LIN {X 0,Y 62.23,Z 1055.519,A -85,B 0,C 180,E1 2367.907,E2 2367.907} C_VEL
LIN {X 0,Y 81.235,Z 1051.075,A -85,B 0,C 180,E1 2356.249,E2 2356.249} C_VEL
LIN {X 0,Y 105.062,Z 1044.254,A -85,B 0,C 180,E1 2348.201,E2 2348.201} C_VEL
LIN {X 0,Y 125.272,Z 1037.346,A -85,B 0,C 180,E1 2343.877,E2 2343.877} C_VEL
LIN {X 0,Y 146.99,Z 1028.752,A -85,B 0,C 180,E1 2340.583,E2 2340.583} C_VEL
LIN {X 0,Y 167.827,Z 1019.239,A -85,B 0,C 180,E1 2338.199,E2 2338.199} C_VEL
LIN {X 0,Y 144.434,Z 1029.702,A -85,B 0,C 180,E1 2335.468,E2 2335.468} C_VEL
LIN {X 0,Y 124.116,Z 1037.572,A -85,B 0,C 180,E1 2332.261,E2 2332.261} C_VEL
LIN {X 0,Y 100.607,Z 1045.395,A -85,B 0,C 180,E1 2326.899,E2 2326.899} C_VEL
LIN {X 0,Y 78.368,Z 1051.328,A -85,B 0,C 180,E1 2318.652,E2 2318.652} C_VEL
LIN {X 0,Y 61.249,Z 1055.193,A -85,B 0,C 180,E1 2307.403,E2 2307.403} C_VEL
LIN {X 0,Y 47.043,Z 1058.07,A -85,B 0,C 180,E1 2288.052,E2 2288.052} C_VEL
LIN {X 0,Y 40.29,Z 1059.695,A -85,B 0,C 180,E1 2260.004,E2 2260.004} C_VEL
LIN {X 0,Y 39.914,Z 1059.95,A -85,B 0,C 180,E1 2244.249,E2 2244.249} C_VEL
LIN {X 0,Y 41.264,Z 1060.011,A -85,B 0,C 180,E1 2225.673,E2 2225.673} C_VEL
LIN {X 0,Y 49.39,Z 1059.265,A -85,B 0,C 180,E1 2201.491,E2 2201.491} C_VEL
LIN {X 0,Y 63.805,Z 1057.416,A -85,B 0,C 180,E1 2184.643,E2 2184.643} C_VEL
LIN {X 0,Y 84.152,Z 1053.993,A -85,B 0,C 180,E1 2173.014,E2 2173.014} C_VEL
LIN {X 0,Y 108.886,Z 1048.344,A -85,B 0,C 180,E1 2165.269,E2 2165.269} C_VEL
LIN {X 0,Y 130.008,Z 1042.364,A -85,B 0,C 180,E1 2161.081,E2 2161.081} C_VEL
LIN {X 0,Y 145.554,Z 1037.228,A -85,B 0,C 180,E1 2158.77,E2 2158.77} C_VEL
LIN {X 0,Y 123.274,Z 1044.544,A -85,B 0,C 180,E1 2155.348,E2 2155.348} C_VEL
LIN {X 0,Y 99.855,Z 1050.86,A -85,B 0,C 180,E1 2150.04,E2 2150.04} C_VEL
LIN {X 0,Y 92.672,Z 1052.424,A -85,B 0,C 180,E1 2148.54,E2 2148.54} C_VEL
LIN {X 0,Y 72.154,Z 1056.236,A -85,B 0,C 180,E1 2145.682,E2 2145.682} C_VEL
LIN {X 0,Y 66.123,Z 1057.108,A -85,B 0,C 180,E1 2143.439,E2 2143.439} C_VEL
LIN {X 0,Y 46.36,Z 1059.586,A -85,B 0,C 180,E1 2127.261,E2 2127.261} C_VEL
LIN {X 0,Y 35.013,Z 1060.577,A -85,B 0,C 180,E1 2102.861,E2 2102.861} C_VEL
LIN {X 0,Y 31.935,Z 1060.688,A -85,B 0,C 180,E1 2077.195,E2 2077.195} C_VEL
LIN {X 0,Y 31.933,Z 1060.508,A -85,B 0,C 180,E1 2062.806,E2 2062.806} C_VEL
LIN {X 0,Y 35.788,Z 1059.542,A -85,B 0,C 180,E1 2034.076,E2 2034.076} C_VEL
LIN {X 0,Y 50.744,Z 1057.023,A -85,B 0,C 180,E1 2007.539,E2 2007.539} C_VEL
LIN {X 0,Y 71.957,Z 1052.634,A -85,B 0,C 180,E1 1993.424,E2 1993.424} C_VEL
LIN {X 0,Y 91.601,Z 1047.732,A -85,B 0,C 180,E1 1986.625,E2 1986.625} C_VEL
LIN {X 0,Y 116.023,Z 1040.405,A -85,B 0,C 180,E1 1981.451,E2 1981.451} C_VEL
LIN {X 0,Y 139.32,Z 1031.761,A -85,B 0,C 180,E1 1978.189,E2 1978.189} C_VEL
LIN {X 0,Y 114.491,Z 1040.77,A -85,B 0,C 180,E1 1974.617,E2 1974.617} C_VEL
LIN {X 0,Y 91.487,Z 1047.54,A -85,B 0,C 180,E1 1969.616,E2 1969.616} C_VEL
LIN {X 0,Y 71.294,Z 1052.467,A -85,B 0,C 180,E1 1962.493,E2 1962.493} C_VEL
LIN {X 0,Y 49.02,Z 1056.839,A -85,B 0,C 180,E1 1946.75,E2 1946.75} C_VEL
LIN {X 0,Y 35.858,Z 1058.993,A -85,B 0,C 180,E1 1921.992,E2 1921.992} C_VEL
LIN {X 0,Y 31.97,Z 1059.896,A -85,B 0,C 180,E1 1893.586,E2 1893.586} C_VEL
LIN {X 0,Y 32.157,Z 1060.129,A -85,B 0,C 180,E1 1875.596,E2 1875.596} C_VEL
LIN {X 0,Y 39.331,Z 1059.836,A -85,B 0,C 180,E1 1842.502,E2 1842.502} C_VEL
LIN {X 0,Y 57.397,Z 1057.92,A -85,B 0,C 180,E1 1819.827,E2 1819.827} C_VEL
LIN {X 0,Y 77.014,Z 1054.988,A -85,B 0,C 180,E1 1809.347,E2 1809.347} C_VEL
LIN {X 0,Y 101.426,Z 1050.147,A -85,B 0,C 180,E1 1802.26,E2 1802.26} C_VEL
LIN {X 0,Y 120.013,Z 1045.405,A -85,B 0,C 180,E1 1798.786,E2 1798.786} C_VEL
LIN {X 0,Y 94.543,Z 1051.731,A -85,B 0,C 180,E1 1793.795,E2 1793.795} C_VEL
LIN {X 0,Y 73.855,Z 1055.787,A -85,B 0,C 180,E1 1787.103,E2 1787.103} C_VEL
LIN {X 0,Y 66.123,Z 1057.108,A -85,B 0,C 180,E1 1783.439,E2 1783.439} C_VEL
LIN {X 0,Y 59.161,Z 1057.998,A -85,B 0,C 180,E1 1780.392,E2 1780.392} C_VEL
LIN {X 0,Y 38.812,Z 1060.018,A -85,B 0,C 180,E1 1771.206,E2 1771.206} C_VEL
LIN {X 0,Y 34.014,Z 1060.279,A -85,B 0,C 180,E1 1765.205,E2 1765.205} C_VEL
LIN {X 0,Y 24.195,Z 1060.648,A -85,B 0,C 180,E1 1724.358,E2 1724.358} C_VEL
LIN {X 0,Y 23.898,Z 1060.472,A -85,B 0,C 180,E1 1705.201,E2 1705.201} C_VEL
LIN {X 0,Y 27.039,Z 1059.798,A -85,B 0,C 180,E1 1673.725,E2 1673.725} C_VEL
LIN {X 0,Y 39.211,Z 1058.087,A -85,B 0,C 180,E1 1646.813,E2 1646.813} C_VEL
LIN {X 0,Y 57.327,Z 1055.125,A -85,B 0,C 180,E1 1632.383,E2 1632.383} C_VEL
LIN {X 0,Y 81.873,Z 1049.995,A -85,B 0,C 180,E1 1623.501,E2 1623.501} C_VEL
LIN {X 0,Y 106.013,Z 1043.342,A -85,B 0,C 180,E1 1618.741,E2 1618.741} C_VEL
LIN {X 0,Y 109.795,Z 1042.185,A -85,B 0,C 180,E1 1618.138,E2 1618.138} C_VEL
LIN {X 0,Y 88.425,Z 1048.176,A -85,B 0,C 180,E1 1614.313,E2 1614.313} C_VEL
LIN {X 0,Y 64.607,Z 1053.606,A -85,B 0,C 180,E1 1607.164,E2 1607.164} C_VEL
LIN {X 0,Y 41.807,Z 1057.387,A -85,B 0,C 180,E1 1592.24,E2 1592.24} C_VEL
LIN {X 0,Y 28.279,Z 1059.218,A -85,B 0,C 180,E1 1566.946,E2 1566.946} C_VEL
LIN {X 0,Y 23.986,Z 1059.979,A -85,B 0,C 180,E1 1534.781,E2 1534.781} C_VEL
LIN {X 0,Y 24.237,Z 1060.188,A -85,B 0,C 180,E1 1513.214,E2 1513.214} C_VEL
LIN {X 0,Y 32.914,Z 1059.953,A -85,B 0,C 180,E1 1474.891,E2 1474.891} C_VEL
LIN {X 0,Y 54.21,Z 1058.087,A -85,B 0,C 180,E1 1452.156,E2 1452.156} C_VEL
LIN {X 0,Y 75.123,Z 1055.192,A -85,B 0,C 180,E1 1443.382,E2 1443.382} C_VEL
LIN {X 0,Y 93.785,Z 1051.742,A -85,B 0,C 180,E1 1438.8,E2 1438.8} C_VEL
LIN {X 0,Y 72.457,Z 1055.741,A -85,B 0,C 180,E1 1433.509,E2 1433.509} C_VEL
LIN {X 0,Y 48.416,Z 1059.029,A -85,B 0,C 180,E1 1421.806,E2 1421.806} C_VEL
LIN {X 0,Y 34.014,Z 1060.279,A -85,B 0,C 180,E1 1405.205,E2 1405.205} C_VEL
LIN {X 0,Y 28.476,Z 1060.509,A -85,B 0,C 180,E1 1395.118,E2 1395.118} C_VEL
LIN {X 0,Y 21.095,Z 1060.68,A -85,B 0,C 180,E1 1377.104,E2 1377.104} C_VEL
LIN {X 0,Y 16.944,Z 1060.254,A -85,B 0,C 180,E1 1322.989,E2 1322.989} C_VEL
LIN {X 0,Y 31.831,Z 1058.564,A -85,B 0,C 180,E1 1279.547,E2 1279.547} C_VEL
LIN {X 0,Y 52.569,Z 1055.608,A -85,B 0,C 180,E1 1265.457,E2 1265.457} C_VEL
LIN {X 0,Y 73.999,Z 1051.54,A -85,B 0,C 180,E1 1259.166,E2 1259.166} C_VEL
LIN {X 0,Y 79.035,Z 1050.485,A -85,B 0,C 180,E1 1258.084,E2 1258.084} C_VEL
LIN {X 0,Y 55.552,Z 1055.004,A -85,B 0,C 180,E1 1251.869,E2 1251.869} C_VEL
LIN {X 0,Y 36.013,Z 1057.824,A -85,B 0,C 180,E1 1240.733,E2 1240.733} C_VEL
LIN {X 0,Y 20.45,Z 1059.511,A -85,B 0,C 180,E1 1213.196,E2 1213.196} C_VEL
LIN {X 0,Y 15.91,Z 1060.107,A -85,B 0,C 180,E1 1169.998,E2 1169.998} C_VEL
LIN {X 0,Y 18.067,Z 1060.358,A -85,B 0,C 180,E1 1132.498,E2 1132.498} C_VEL
LIN {X 0,Y 35.082,Z 1059.66,A -85,B 0,C 180,E1 1094.289,E2 1094.289} C_VEL
LIN {X 0,Y 56.034,Z 1057.808,A -85,B 0,C 180,E1 1082.17,E2 1082.17} C_VEL
LIN {X 0,Y 66.796,Z 1056.536,A -85,B 0,C 180,E1 1078.887,E2 1078.887} C_VEL
LIN {X 0,Y 41.792,Z 1059.315,A -85,B 0,C 180,E1 1068.795,E2 1068.795} C_VEL
LIN {X 0,Y 23.803,Z 1060.403,A -85,B 0,C 180,E1 1047.156,E2 1047.156} C_VEL
LIN {X 0,Y 16.114,Z 1060.522,A -85,B 0,C 180,E1 1004.372,E2 1004.372} C_VEL
LIN {X 0,Y 15.989,Z 1060.366,A -85,B 0,C 180,E1 979.189,E2 979.189} C_VEL
LIN {X 0,Y 16.944,Z 1060.254,A -85,B 0,C 180,E1 962.989,E2 962.989} C_VEL
LIN {X 0,Y 19.569,Z 1059.953,A -85,B 0,C 180,E1 941.806,E2 941.806} C_VEL
LIN {X 0,Y 26.288,Z 1059.023,A -85,B 0,C 180,E1 915.615,E2 915.615} C_VEL
LIN {X 0,Y 35.66,Z 1057.813,A -85,B 0,C 180,E1 902.3,E2 902.3} C_VEL
LIN {X 0,Y 39.85,Z 1057.312,A -85,B 0,C 180,E1 900.013,E2 900.013} C_VEL
LIN {X 0,Y 45.651,Z 1056.586,A -85,B 0,C 180,E1 898.004,E2 898.004} C_VEL
LIN {X 0,Y 21.184,Z 1059.185,A -85,B 0,C 180,E1 883.548,E2 883.548} C_VEL
LIN {X 0,Y 8.405,Z 1060.123,A -85,B 0,C 180,E1 830.907,E2 830.907} C_VEL
LIN {X 0,Y 8.481,Z 1060.284,A -85,B 0,C 180,E1 781.86,E2 781.86} C_VEL
LIN {X 0,Y 21.347,Z 1060.227,A -85,B 0,C 180,E1 730.374,E2 730.374} C_VEL
LIN {X 0,Y 37.624,Z 1059.486,A -85,B 0,C 180,E1 718.952,E2 718.952} C_VEL
LIN {X 0,Y 18.721,Z 1060.378,A -85,B 0,C 180,E1 704.025,E2 704.025} C_VEL
LIN {X 0,Y 8.236,Z 1060.418,A -85,B 0,C 180,E1 651.362,E2 651.362} C_VEL
LIN {X 0,Y 8.234,Z 1060.283,A -85,B 0,C 180,E1 608.638,E2 608.638} C_VEL
LIN {X 0,Y 21.469,Z 1059.26,A -85,B 0,C 180,E1 552.034,E2 552.034} C_VEL
LIN {X 0,Y 39.85,Z 1057.312,A -85,B 0,C 180,E1 540.013,E2 540.013} C_VEL
LIN {X 0,Y 42.01,Z 1059.299,A -85,B 0,C 180,E1 539.267,E2 539.267} C_VEL
LIN {X 0,Y 42.01,Z 1075.5,A -85,B 0,C 180,E1 539.267,E2 539.267} C_VEL
LIN {X 0,Y 42.01,Z 1075.5,A -85,B 0,C 180,E1 539.267,E2 539.267}

QRS_NEXT_CUT()

QRS_NEXT()
QRS_HOME()

END
